TYPE ST_Robot :
STRUCT
    id           : DINT;
    name         : STRING(80);
    manufacturer : STRING(80);
    model        : STRING(80);
    robot_type   : STRING(80);
    axes         : DINT;
    payload      : LREAL;
    reach        : LREAL;
    controller   : STRING(80);
    ip_address   : STRING(40);
END_STRUCT
END_TYPE

(* stored: Version 1.1.0.1, ProductVersion 3.1.4026.18
   DUT ST_Robot: Id {cfce4933-d5fc-4925-b85d-aea37258ed8b} *)
